(*
SPDX-FileCopyrightText: © 2026 Oleksandr Tiutyk <trofimich@gmail.com>
SPDX-License-Identifier: MIT
License: https://opensource.org/license/mit
*)

(*!
<summary>Provides lookup and indexed access to a collection of unique generic values.</summary>
<description>
Generic query descriptors are borrowed by default. Explicit release disposes only owned query storage and does
not reset caller-side aliases. The source collection and borrowed payload must remain alive while returned
references are used; mutation can invalidate positions and references. Lookup uses one equality/hash strategy
fixed for the collection lifetime; zero selects GENERIC_VALUE default equality and hashing. A custom comparer
is borrowed, stays alive and retains stable equality-relevant configuration. Empty descriptors are supported
unless rejected by a validator. No entry or enumeration order is guaranteed; a position is a current storage
slot, not a sorted rank. Do not modify stored descriptors through returned references. Borrowed elements,
including OBJECT instances, stay alive while stored and remain caller-owned. Owned payload must not be deleted
through external aliases. Keep equality/hash-relevant data and comparer configuration stable; remove before
changing them, then insert again. Fields unrelated to equality/hash may change. Callbacks must not mutate
elements or reenter collection mutation. Explicit query release must not dispose of retained storage. Default
OBJECT lookup delegates to Object.Equals/GetHashCode; Clone has its own identity. Discard and populate the
index again after equality-relevant address relocation before further lookup.
</description>
*)
INTERFACE IReadOnlyUniqueDataSet EXTENDS ICollection

(*!
<summary>Reports whether a matching raw query exists.</summary>
<description>
The raw ANY argument is borrowed without cloning or ownership transfer. isObject = TRUE requires a live Object
function-block instance, not a pointer or interface variable. FALSE uses ordinary runtime type mapping. The
caller keeps the query storage alive for the call.
</description>
*)
//!<param name="isObject">Explicitly interprets the raw argument as a live Object instance.</param>
METHOD Contains : BOOL
VAR_INPUT
	value : ANY;
	isObject : BOOL := FALSE;
END_VAR
END_METHOD

(*!
<summary>Reports whether a matching entry exists for a borrowed generic query.</summary>
<description>
The query is borrowed by default. Explicit release requests disposal of owned query storage after lookup
completes, including a missing result. Requested release is attempted after both successful lookup and lookup
failure. Before cleanup, the original framework exception is retained and a borrowed static system exception
is cloned to preserve its code, catch point and timestamps across cleanup callbacks. The captured exception is
then propagated through ExceptionManager.Throw in the current cyclic task; native errors use the framework
SystemException representation. If capturing the system exception fails with terminal OOM, query cleanup is
still attempted and terminal OOM takes precedence. Terminal allocation state is never cleared. Release is best
effort and does not prove successful deallocation. Cleanup callbacks must not reenter collection mutation.
Release resets only the local descriptor copy; the caller must have disposal rights and must not reuse or
release owning aliases afterwards. Borrowed payload is not freed.
</description>
*)
METHOD ContainsGeneric : BOOL
VAR_INPUT
	value : TOF_Core.GENERIC_VALUE;
	releaseValue : BOOL := FALSE;
END_VAR
END_METHOD

(*!
<summary>Borrows the entry at a current storage position.</summary>
<description>
The index must be within Length and is not a sorted rank; otherwise an exception is raised. The returned
descriptor reference and payload remain collection-owned or borrowed from their original owner. Do not mutate
the descriptor or dispose of its payload through this view. Mutation or destruction may invalidate the
reference.
</description>
*)
METHOD GetByIndex : REFERENCE TO TOF_Core.GENERIC_VALUE
VAR_INPUT
	index : DINT;
END_VAR
END_METHOD

(*!
<summary>Returns the matching entry position, or a negative value when absent.</summary>
<description>
The query is borrowed by default. Explicit release requests disposal of owned query storage after lookup
completes, including a missing result. Requested release is attempted after both successful lookup and lookup
failure. Before cleanup, the original framework exception is retained and a borrowed static system exception
is cloned to preserve its code, catch point and timestamps across cleanup callbacks. The captured exception is
then propagated through ExceptionManager.Throw in the current cyclic task; native errors use the framework
SystemException representation. If capturing the system exception fails with terminal OOM, query cleanup is
still attempted and terminal OOM takes precedence. Terminal allocation state is never cleared. Release is best
effort and does not prove successful deallocation. Cleanup callbacks must not reenter collection mutation.
Release resets only the local descriptor copy; the caller must have disposal rights and must not reuse or
release owning aliases afterwards. Borrowed payload is not freed. The position is a current storage slot with
no sorted-rank guarantee; mutation may invalidate it.
</description>
*)
METHOD GetGenericValuePosition : DINT
VAR_INPUT
	value : TOF_Core.GENERIC_VALUE;
	releaseValue : BOOL := FALSE;
END_VAR
END_METHOD

(*!
<summary>Returns the matching storage position, or a negative value when absent.</summary>
<description>
The raw ANY argument is borrowed without cloning or ownership transfer. isObject = TRUE requires a live Object
function-block instance, not a pointer or interface variable. FALSE uses ordinary runtime type mapping. The
caller keeps the query storage alive for the call. The position is a current storage slot with no sorted-rank
guarantee; mutation may invalidate it.
</description>
*)
//!<param name="isObject">Explicitly interprets the raw argument as a live Object instance.</param>
METHOD GetValuePosition : DINT
VAR_INPUT
	value : ANY;
	isObject : BOOL := FALSE;
END_VAR
END_METHOD

END_INTERFACE

(* stored: Version 1.1.0.1
   Itf IReadOnlyUniqueDataSet: Id {ed37f372-aa88-4c4c-9aad-3bf978f2dfed}
   Method Contains: Id {e115c275-76c1-4f4d-8997-0776645d585b}
   Method ContainsGeneric: Id {74cd7913-6f9d-4999-a0d9-9e406cf5bb6a}
   Method GetByIndex: Id {25bc667f-4f18-44ec-8341-f0e780ab0dbf}
   Method GetGenericValuePosition: Id {125f3f63-b0f5-4242-b588-4edd1f9b6ae2}
   Method GetValuePosition: Id {f5c205a1-0211-4b4d-9dbb-b510491d9cbf} *)
